FUNCTION_BLOCK DigitalSignal
VAR_INPUT
	Signal: BOOL;
END_VAR
VAR_OUTPUT
	State: BOOL;
END_VAR
VAR
	_PosFlank: BOOL;
	_NegFlank: BOOL;
	OffTimer: Timer;
	OnTimer: Timer;
END_VAR

IF Signal <> State THEN
	State := Signal;
	IF State THEN
	  _PosFlank := TRUE;
	ELSE
	  _NegFlank := TRUE;
	END_IF;
END_IF;
IF State THEN
	OffTimer.Restart();
ELSE
	OnTimer.Restart();
END_IF

METHOD NegFlank : BOOL
VAR_INPUT
	Reset: BOOL;
END_VAR
NegFlank := _NegFlank;
if Reset then
	_NegFlank := FALSE;
END_IF
END_METHOD

METHOD OffTime : LINT
VAR_INPUT
END_VAR
IF State THEN
	OffTimer.Restart();
ELSE
	OnTimer.Restart();
END_IF
OffTime := OffTimer.ElapsedTime();
END_METHOD

METHOD OnTime : LINT
VAR_INPUT
END_VAR
IF State THEN
	OffTimer.Restart();
ELSE
	OnTimer.Restart();
END_IF
OnTime := OnTimer.ElapsedTime();
END_METHOD

METHOD PosFlank : BOOL
VAR_INPUT
	Reset: BOOL := FALSE;
END_VAR
PosFlank := _PosFlank;
if Reset then
	_PosFlank := FALSE;
END_IF
END_METHOD

END_FUNCTION_BLOCK

(* stored: Version 1.1.0.1, ProductVersion 3.1.4024.6
   POU DigitalSignal: Id {479e134f-75f0-4165-808c-efafb9f88e44}, SpecialFunc None
   Method NegFlank: Id {084ad7ff-3517-4efc-bf51-73b1040e8e50}
   Method OffTime: Id {6870f297-3563-48d6-a194-4c0a89294c1a}
   Method OnTime: Id {737c220b-e6d8-4cd6-9d85-6e4160018fd8}
   Method PosFlank: Id {71808a80-b9c8-4ffa-a24c-b4dc129a17f1} *)
